// Mitsubishi GX Works2 project: 아날로그 속도 제어   PLC: Q03UDV

PROGRAM MAIN
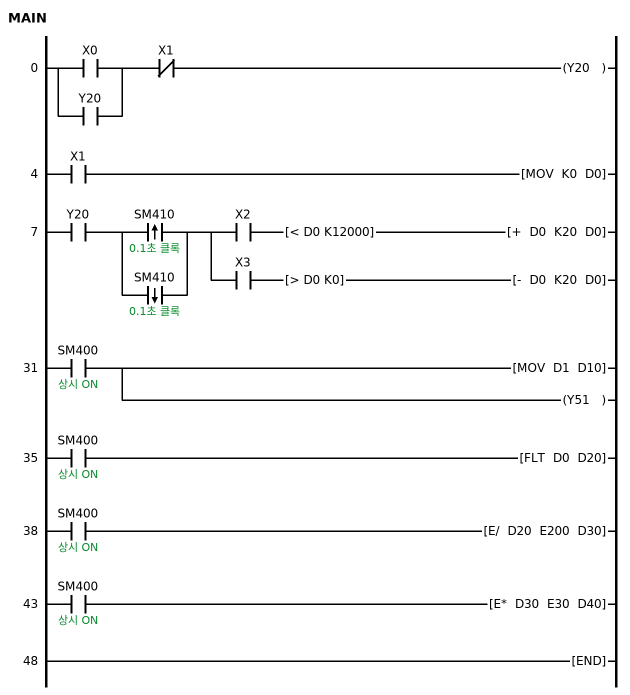
0     LD      X0
      OR      Y20
      ANI     X1
      OUT     Y20
4     LD      X1
      MOV     K0 D0
7     LD      Y20
      LDP     SM410  ; 0.1초 클록
      ORF     SM410  ; 0.1초 클록
      ANB
      MPS
      AND     X2
      AND<    D0 K12000
      +       D0 K20 D0
      MPP
      AND     X3
      AND>    D0 K0
      -       D0 K20 D0
31    LD      SM400  ; 상시 ON
      MOV     D1 D10
      OUT     Y51
35    LD      SM400  ; 상시 ON
      FLT     D0 D20
38    LD      SM400  ; 상시 ON
      E/      D20 E200 D30
43    LD      SM400  ; 상시 ON
      E*      D30 E30 D40
48    END
END_PROGRAM
